(*			
	EVERDE sp. z o.o.
	Rafał Osajda		08.08.2025		TC 4024.66
	Interfejs do wyciągania z SPM przez HMI danych do wyświetlania - dla okna PUSTE
*)
INTERFACE ITF_SPM_HMI_Pusty_Lacznik EXTENDS  B_Baza.ITF_ZrodloIdentyfikacji

END_INTERFACE

(* stored: Version 1.1.0.1
   Itf ITF_SPM_HMI_Pusty_Lacznik: Id {2c4b4f1b-43cc-0c56-25bf-78791c2e26d4} *)
